// TIA Portal V18 export
// export: Created 2025-12-01T17:52:55.8885707Z, ExportSetting None, DisplayName Totally Integrated Automation Portal, DisplayVersion V18 Update 5, DisplayName TIA Portal Openness, DisplayVersion V18 Update 5, DisplayName TIA Portal Teamcenter Gateway, DisplayVersion V18, DisplayName TIA Portal Version Control Interface, DisplayVersion V18, DisplayName STEP 7 Professional, DisplayVersion V18 Update 5, DisplayName STEP 7 Safety, DisplayVersion V18, DisplayName WinCC Professional, DisplayVersion V18 Update 5
Screen "130 Process Data Layout"  1280x800, Number=11, Template=00MainScreen
  on GenerateScreen: SetBit(Tag := NormalON); ResetBit(Tag := NormalOFF); SetTag(Tag := ST_SysDBNum, Value := 1060); SetTag(Tag := PM_CountCycleDBNum, Value := 1061); SetTag(Tag := ST_PMDBNum, Value := 1063)
  ScreenLayer 
    Button "按钮_4" at 383,725 size 128x75  PictureOff=向右箭头_0, StyleItem=BtnNormal20, TextOff="报 警 / Alarm / Poplach"
      RangeAppearanceAnimation "RangeAppearanceAnimation"
        tag ST_AlarmON
        1..1: back #ff0000, fore #d6d3ce, flashing
      on Click: ActivateScreen(Screen name := 300Main, Object number := 0); SetTag(Tag := Sys_VersionManagement_HMIPageID, Value := 300)
    Button "按钮_6"  Authorization=Manage Parameter, PictureOff=向右箭头_0, StyleItem=BtnNormal20, TextOff="参数设定 / Parameter setting / Parameter nastavenie", TextOn="参数设定 / Parameter setting / Parameter nastavenie"
      RangeAppearanceAnimation "RangeAppearanceAnimation"
        tag _unlock[5]
        0..0: back #d6e1e8, fore #c0c0c0
      on Click: ActivateScreen(Screen name := 700 Main, Object number := 0)
    Button "按钮_8" at 511,725 size 128x75  StyleItem=BtnNormal20, TextOff="MES", TextOn="照明灯 / Light / Svetlo"
      on Press: ActivateScreen(Screen name := 900MES, Object number := 0); SetTag(Tag := Sys_VersionManagement_HMIPageID, Value := 900)
    Button "按钮_11" at 256,725 size 128x75  PictureOff=向右箭头_0, StyleItem=BtnNormal20, TextOff="Safety Status", TextOn="Safety Status"
      on Click: ShowPopupScreen(Name of the screen := Pilz, X coordinate := 350, Y coordinate := 150, Display mode := -1, Animation := -1, Animation speed := 1)
    Button "btnMenu5_1" at 128,725 size 128x75  StyleItem=BtnNormal22, TextOff="主页面 / Main", TextOn="主页面 / Main"
      on Click: ActivateScreen(Screen name := , Object number := 0); SetTag(Tag := Sys_VersionManagement_HMIPageID, Value := 10)
    Button "按钮_1"  PictureOff=向右箭头_0, StyleItem=BtnNormal20, TextList=蜂鸣器屏蔽, TextOff="蜂鸣器 屏蔽 / Buzzer shield / Bzučiak štít", TextOn="蜂鸣器 屏蔽 / Buzzer shield"
      RangeAppearanceAnimation "RangeAppearanceAnimation"
        tag ST_CommandBuzzerOn
        1..1: back #3366ff, fore #d6d3ce
      on Click: InvertBit(Tag := ST_CommandBuzzerOn)
      ProcessValue := ST_CommandBuzzerOn
    Circle "圆_1" at 259,725 size 29x29
      RangeAppearanceAnimation "RangeAppearanceAnimation"
        tag PilzData_Status
        1..1: back #00ff00, fore #181c31
        2..2: back #ff0000, fore #181c31
    TextField "Template_Text field_1" at 855,4 size 299x25  Text="Tool scanning code is running"
      RangeAppearanceAnimation "RangeAppearanceAnimation"
        tag ChangeOver_DB_Global_ScanFixtureFlag
        1..1: back #00ff00, fore #31344a, flashing
      SingleBitVisibilityAnimation "VisibilityAnimation"
        tag ChangeOver_DB_Global_ScanFixtureFlag
    Button "按钮_2"  StyleItem=BtnNormal20, TextOff="清料模式 / Empty Mode / Text", TextOn="清料模式 / Clearing Mode / Text"
      RangeAppearanceAnimation "RangeAppearanceAnimation"
        tag AutoProcessControl_Robot_1_ClearPart
        0..0: back #d6e1e8, fore #000000
        1..1: back #00ff00, fore #000000
      on Click: InvertBit(Tag := AutoProcessControl_Robot_1_ClearPart)
    Button "btnMenu7_6" at 767,725 size 128x75  StyleItem=BtnNormal20
    Button "btnMenu7_15" at 639,725 size 128x75  StyleItem=BtnActive18, TextOff="Process data Layout", TextOn="Process data Layout"
      on Click: ActivateScreen(Screen name := , Object number := 0)
  ScreenLayer 
    GraphicView "图形视图_1" at 205,98 size 972x584  Picture=图形_44
  ScreenLayer 
    Button "btnMenu7_23" at 907,500 size 123x49  TextOff="E-NG盒2 / GLUE NG Buffer / E-NG2", TextOn="E-NG盒2 / E-NG2"
      on Click: SetTag(Tag := AutoProcess_HMI_IndexProcess, Value := 0); ShowPopupScreen(Name of the screen := AutoProcessDataPopUp, X coordinate := 280, Y coordinate := 100, Display mode := 1, Animation := 3, Animation speed := 2)
    Button "btnMenu7_4" at 626,583 size 119x36  TextOff="B-压机2 / B-Press2", TextOn="B-压机2 / B-Press2"
      on Click: SetTag(Tag := AutoProcess_HMI_IndexProcess, Value := 10); ShowPopupScreen(Name of the screen := AutoProcessDataPopUp, X coordinate := 280, Y coordinate := 100, Display mode := 1, Animation := 3, Animation speed := 2)
    Button "btnMenu7_22" at 703,261 size 129x35  TextOff="F-机器人3 / F-Robot3", TextOn="F-机器人3 / F-Robot3"
      on Click: SetTag(Tag := AutoProcess_HMI_IndexProcess, Value := 11); ShowPopupScreen(Name of the screen := AutoProcessDataPopUp, X coordinate := 280, Y coordinate := 100, Display mode := 1, Animation := 3, Animation speed := 2)
    Button "btnMenu7_21" at 526,261 size 127x35  TextOff="F-机器人2 / F-Robot2", TextOn="F-机器人2 / F-Robot2"
      on Click: SetTag(Tag := AutoProcess_HMI_IndexProcess, Value := 6); ShowPopupScreen(Name of the screen := AutoProcessDataPopUp, X coordinate := 280, Y coordinate := 100, Display mode := 1, Animation := 3, Animation speed := 2)
    Button "btnMenu7_3" at 518,572 size 104x38  TextOff="C-Glue", TextOn="C-Glue"
      on Click: SetTag(Tag := AutoProcess_HMI_IndexProcess, Value := 5); ShowPopupScreen(Name of the screen := AutoProcessDataPopUp, X coordinate := 280, Y coordinate := 100, Display mode := 1, Animation := 3, Animation speed := 2)
    Button "btnMenu7_1" at 360,558 size 113x37  TextOff="B-压机1 / B-Press1", TextOn="B-压机1 / B-Press1"
      on Click: SetTag(Tag := AutoProcess_HMI_IndexProcess, Value := 4); ShowPopupScreen(Name of the screen := AutoProcessDataPopUp, X coordinate := 280, Y coordinate := 100, Display mode := 1, Animation := 3, Animation speed := 2)
    Button "btnMenu7_2" at 232,555 size 124x46  TextOff="A-Ring1 上料 / A - scan rotate / A-Load Ring1", TextOn="A-Ring1 上料 / A-Load Ring1"
      on Click: SetTag(Tag := AutoProcess_HMI_IndexProcess, Value := 1); ShowPopupScreen(Name of the screen := AutoProcessDataPopUp, X coordinate := 280, Y coordinate := 100, Display mode := 1, Animation := 3, Animation speed := 2)
    Button "btnMenu7_24" at 144,443 size 141x49  TextOff="E-NG盒1 / Magn Scan NG Buffer / E-NG1", TextOn="E-NG盒1 / E-NG1"
      on Click: SetTag(Tag := AutoProcess_HMI_IndexProcess, Value := 9); ShowPopupScreen(Name of the screen := AutoProcessDataPopUp, X coordinate := 280, Y coordinate := 100, Display mode := 1, Animation := 3, Animation speed := 2)
    Button "btnMenu7_20" at 308,261 size 146x35  TextOff="F-机器人1 / Rob1-shaft / F-Robot1", TextOn="F-机器人1 / F-Robot1"
      on Click: SetTag(Tag := AutoProcess_HMI_IndexProcess, Value := 2); ShowPopupScreen(Name of the screen := AutoProcessDataPopUp, X coordinate := 280, Y coordinate := 100, Display mode := 1, Animation := 3, Animation speed := 2)
    Button "btnMenu7_12" at 268,100 size 140x35  TextOff="H- 轴上料 / H-ShaftBelt / H- ShaftBelt", TextOn="H- 轴上料 / H- ShaftBelt"
      on Click: SetTag(Tag := AutoProcess_HMI_IndexProcess, Value := 13); ShowPopupScreen(Name of the screen := AutoProcessDataPopUp, X coordinate := 280, Y coordinate := 100, Display mode := 1, Animation := 3, Animation speed := 2)
    Button "btnMenu7_16" at 444,100 size 156x35  TextOff="J- 磁铁上料 / J-MagnetBelt / J- MagnetBelt", TextOn="J- 磁铁上料 / J- MagnetBelt"
      on Click: SetTag(Tag := AutoProcess_HMI_IndexProcess, Value := 14); ShowPopupScreen(Name of the screen := AutoProcessDataPopUp, X coordinate := 280, Y coordinate := 100, Display mode := 1, Animation := 3, Animation speed := 2)
    Button "btnMenu7_17" at 616,100 size 162x35  TextOff="K-预留 上料//预留 / K-ReserveBelt / K- ReserveBelt", TextOn="K-预留 上料//预留 / K- ReserveBelt"
      on Click: SetTag(Tag := AutoProcess_HMI_IndexProcess, Value := 15); ShowPopupScreen(Name of the screen := AutoProcessDataPopUp, X coordinate := 280, Y coordinate := 100, Display mode := 1, Animation := 3, Animation speed := 2)
    Button "btnMenu7_18" at 785,100 size 153x35  TextOff="L- 空托盘 / L-UnloadBelt / L- UnloadBelt", TextOn="L- 空托盘 / L- UnloadBelt"
      on Click: SetTag(Tag := AutoProcess_HMI_IndexProcess, Value := 16); ShowPopupScreen(Name of the screen := AutoProcessDataPopUp, X coordinate := 280, Y coordinate := 100, Display mode := 1, Animation := 3, Animation speed := 2)
    Button "btnMenu7_7" at 703,301 size 129x35  TextOff="F-机器人3 / F-Robot3", TextOn="F-机器人3 / F-Robot3"
      on Click: SetTag(Tag := AutoProcess_HMI_IndexProcess, Value := 12); ShowPopupScreen(Name of the screen := AutoProcessDataPopUp, X coordinate := 280, Y coordinate := 100, Display mode := 1, Animation := 3, Animation speed := 2)
    Button "btnMenu7_8" at 526,301 size 127x35  TextOff="F-机器人2 / F-Robot2", TextOn="F-机器人2 / F-Robot2"
      on Click: SetTag(Tag := AutoProcess_HMI_IndexProcess, Value := 7); ShowPopupScreen(Name of the screen := AutoProcessDataPopUp, X coordinate := 280, Y coordinate := 100, Display mode := 1, Animation := 3, Animation speed := 2)
    Button "btnMenu7_9" at 308,301 size 138x35  TextOff="F-机器人1 / Rob1-Ring / F-Robot1", TextOn="F-机器人1 / F-Robot1"
      on Click: SetTag(Tag := AutoProcess_HMI_IndexProcess, Value := 3); ShowPopupScreen(Name of the screen := AutoProcessDataPopUp, X coordinate := 280, Y coordinate := 100, Display mode := 1, Animation := 3, Animation speed := 2)
  ScreenLayer 
    GraphicIOField "图形 I/O 域_4" at 786,101 size 36x33  Mode=Output, PictureList=productpresent
      ProcessValue := AutoProcess_HMI_StationHasProduct{16}
    GraphicIOField "图形 I/O 域_3" at 617,101 size 36x33  Mode=Output, PictureList=productpresent
      ProcessValue := AutoProcess_HMI_StationHasProduct{15}
    GraphicIOField "图形 I/O 域_2" at 445,101 size 36x33  Mode=Output, PictureList=productpresent
      ProcessValue := AutoProcess_HMI_StationHasProduct{14}
    GraphicIOField "图形 I/O 域_1" at 270,101 size 36x33  Mode=Output, PictureList=productpresent
      ProcessValue := AutoProcess_HMI_StationHasProduct{13}
    GraphicIOField "图形 I/O 域_6" at 309,262 size 36x33  Mode=Output, PictureList=productpresent
      ProcessValue := AutoProcess_HMI_StationHasProduct{2}
    GraphicIOField "图形 I/O 域_11" at 145,452 size 36x33  Mode=Output, PictureList=productpresent
      ProcessValue := AutoProcess_HMI_StationHasProduct{9}
    GraphicIOField "图形 I/O 域_9" at 233,561 size 36x33  Mode=Output, PictureList=productpresent
      ProcessValue := AutoProcess_HMI_StationHasProduct{1}
    GraphicIOField "图形 I/O 域_12" at 361,560 size 36x33  Mode=Output, PictureList=productpresent
      ProcessValue := AutoProcess_HMI_StationHasProduct{4}
    GraphicIOField "图形 I/O 域_15" at 519,574 size 36x33  Mode=Output, PictureList=productpresent
      ProcessValue := AutoProcess_HMI_StationHasProduct{5}
    GraphicIOField "图形 I/O 域_7" at 527,262 size 36x33  Mode=Output, PictureList=productpresent
      ProcessValue := AutoProcess_HMI_StationHasProduct{6}
    GraphicIOField "图形 I/O 域_8" at 704,262 size 36x33  Mode=Output, PictureList=productpresent
      ProcessValue := AutoProcess_HMI_StationHasProduct{11}
    GraphicIOField "图形 I/O 域_13" at 627,584 size 36x33  Mode=Output, PictureList=productpresent
      ProcessValue := AutoProcess_HMI_StationHasProduct{10}
    GraphicIOField "图形 I/O 域_10" at 908,508 size 36x33  Mode=Output, PictureList=productpresent
      ProcessValue := AutoProcess_HMI_StationHasProduct{8}
    GraphicIOField "图形 I/O 域_5" at 309,302 size 36x33  Mode=Output, PictureList=productpresent
      ProcessValue := AutoProcess_HMI_StationHasProduct{3}
    GraphicIOField "图形 I/O 域_16" at 527,302 size 36x33  Mode=Output, PictureList=productpresent
      ProcessValue := AutoProcess_HMI_StationHasProduct{7}
    GraphicIOField "图形 I/O 域_17" at 704,302 size 36x33  Mode=Output, PictureList=productpresent
      ProcessValue := AutoProcess_HMI_StationHasProduct{12}
